PROGRAM pouDPDiag
VAR
	i: UINT;
END_VAR
VAR // added by the converter: edge detectors and wires of the graphical bodies
    _rt1 : R_TRIG;
END_VAR

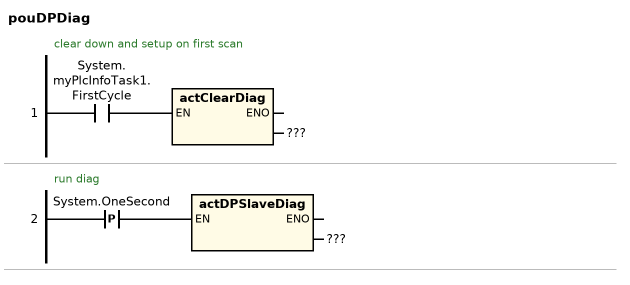
// NETWORK 1
// clear down and setup on first scan
IF System.myPlcInfoTask1.FirstCycle THEN actClearDiag(); END_IF

// NETWORK 2
// run diag
_rt1(CLK := System.OneSecond);
IF _rt1.Q THEN actDPSlaveDiag(); END_IF

ACTION actClearDiag:
FOR i := 1 TO profibusDiag.maxNumDPSlaves DO
	
	//clear memory
	profibusDiag.DPslaveDiag[i].currentState := 0;
	profibusDiag.DPslaveDiag[i].historicalState := 0;
	
	//assign slave number
	profibusDiag.DPslaveDiag[i].SlaveNumber := i;
	
	
END_FOR
END_ACTION

ACTION actDPSlaveDiag:
FOR i := 1 TO profibusDiag.maxNumDPSlaves DO
	
	//record outer box
	//record previous state, latching 
	IF profibusDiag.RawDPStateDiag[i] = 0 AND 
	   profibusDiag.DPslaveDiag[i].currentState <> HMIColour.colourGreyBackground AND 
	   profibusDiag.DPslaveDiag[i].historicalState = HMIColour.colourGreyBackground THEN
		//at this time, record the current state in the historical state
		profibusDiag.DPslaveDiag[i].historicalState := profibusDiag.DPslaveDiag[i].currentState;
	END_IF
	
	//clear inner box when fault is resolved
	IF profibusDiag.RawDPStateDiag[i] = 0 AND 
	   gHMIButtons.btnReset THEN
	   profibusDiag.DPslaveDiag[i].historicalState := HMIColour.colourGreyBackground;
	END_IF
	
	//from the profibus DPState word, colour the box
	CASE profibusDiag.RawDPStateDiag[i] OF 
    0	: 	profibusDiag.DPslaveDiag[i].currentState := HMIColour.colourGreyBackground;
			
    1	: 	profibusDiag.DPslaveDiag[i].currentState := HMIColour.colourRed;
	2	: 	profibusDiag.DPslaveDiag[i].currentState := HMIColour.colourRed;
	3	: 	profibusDiag.DPslaveDiag[i].currentState := HMIColour.colourRed;
 	4	: 	profibusDiag.DPslaveDiag[i].currentState := HMIColour.colourRed;
  	5	: 	profibusDiag.DPslaveDiag[i].currentState := HMIColour.colourRed;
  	6	: 	profibusDiag.DPslaveDiag[i].currentState := HMIColour.colourRed;
  	7	: 	profibusDiag.DPslaveDiag[i].currentState := HMIColour.colourRed;
 	8	: 	profibusDiag.DPslaveDiag[i].currentState := HMIColour.colourRed;
 	9	: 	profibusDiag.DPslaveDiag[i].currentState := HMIColour.colourRed;
 	10	: 	profibusDiag.DPslaveDiag[i].currentState := HMIColour.colourRed;
  	11	: 	profibusDiag.DPslaveDiag[i].currentState := HMIColour.colourRed;
  	12	: 	profibusDiag.DPslaveDiag[i].currentState := HMIColour.colourRed;
 	13	: 	profibusDiag.DPslaveDiag[i].currentState := HMIColour.colourRed;
 	14	: 	profibusDiag.DPslaveDiag[i].currentState := HMIColour.colourRed;
 	15	: 	profibusDiag.DPslaveDiag[i].currentState := HMIColour.colourRed;
	16	: 	profibusDiag.DPslaveDiag[i].currentState := HMIColour.colourRed;
	17	: 	profibusDiag.DPslaveDiag[i].currentState := HMIColour.colourRed;
	18	: 	profibusDiag.DPslaveDiag[i].currentState := HMIColour.colourRed;
	
	31	: 	profibusDiag.DPslaveDiag[i].currentState := HMIColour.colourRed;
	
	128	: 	profibusDiag.DPslaveDiag[i].currentState := HMIColour.colourRed;
	129	: 	profibusDiag.DPslaveDiag[i].currentState := HMIColour.colourRed;
	130	: 	profibusDiag.DPslaveDiag[i].currentState := HMIColour.colourRed;
	131	: 	profibusDiag.DPslaveDiag[i].currentState := HMIColour.colourRed;
	132	: 	profibusDiag.DPslaveDiag[i].currentState := HMIColour.colourRed;
					
	
ELSE 
		//invalid state
         profibusDiag.DPslaveDiag[i].currentState := HMIColour.colourPink;
END_CASE;
	
	
	
END_FOR



//taken from help file
//USINT
//0 = No error
//1 = Station deactivated
//2 = Station not exists
//3 = Master lock
//4 = Invalid slave response
//5 = Parameter fault
//6 = Not supported
//7 = Config fault
//8 = Station not ready
//9 = Static diagnosis
//10 = Diagnosis overflow
//11 = Physical fault
//12 = Data-Exchange left
//13 = Severe bus fault
//14 = Telegram fault
//15 = Station has no ressources
//16 = Service not activated
//17 = Unexpected telegram
//18 = Station ready
//31 = only for EtherCAT gateways: WC-State of cyclic EtherCAT frame is 1
//128 = slave, waiting for data transfer (or DP-Master in CLEAR-Mode)
//129	= slave, waiting for configuration
//130	= slave, waiting for parameter
//131	= slave, waiting for baudrate
//132	= slave, waiting for station no. from PLC
END_ACTION

END_PROGRAM

(* stored: Version 1.1.0.1, ProductVersion 3.1.4024.12
   POU pouDPDiag: Id {060421ca-a6ea-4bfb-924e-d88a8c129e51}, SpecialFunc None
   Action actClearDiag: Id {a604ee79-29e9-4188-ad60-31af404e8db1}
   Action actDPSlaveDiag: Id {c5c6f67f-2bb7-4887-a33c-c090b28b9205} *)
